PROGRAM MAIN
VAR
END_VAR

END_PROGRAM

(* stored: Version 1.1.0.1
   POU MAIN: Id {8bb72742-67c8-4792-84ae-e6940c27cae2} *)
